{attribute 'qualified_only'}
{attribute 'strict'}
TYPE E_StrategyType :
(
	HeavyWash,
	NormalWash,
	SoftWash,
	None
);
END_TYPE

(* stored: Version 1.1.0.1, ProductVersion 3.1.4024.16
   DUT E_StrategyType: Id {4d6497f7-ebae-4371-aa94-56c88ae39c2c} *)
